DATA_BLOCK "DT-Chars_DB"
{ S7_Optimized_Access := 'FALSE' }
VERSION : 0.1
NON_RETAIN
// ATTRIBUTES
// AUTO_NUMBER = False
// BLOCK_NUMBER = 2360
// END_ATTRIBUTES
"DT-Chars"

BEGIN

END_DATA_BLOCK

